PROGRAM Motor_Control
VAR
	Start_Stop_0: Start_Stop;
	Trapizoidal_0: Trapizoidal;
	Trapizoidal_1: Trapizoidal;
	BLINK_0: BLINK;
	R_TRIG_0: R_TRIG;
	
	Timer : BOOL;
END_VAR

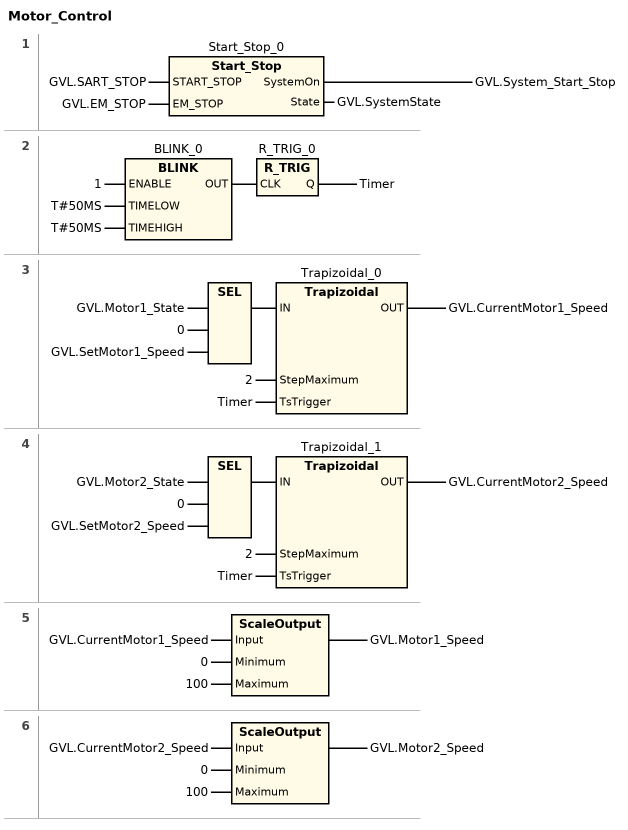
// NETWORK 1
Start_Stop_0(START_STOP := GVL.SART_STOP, EM_STOP := GVL.EM_STOP, State => GVL.SystemState); // Start_Stop
GVL.System_Start_Stop := Start_Stop_0.SystemOn;

// NETWORK 2
BLINK_0(ENABLE := 1, TIMELOW := T#50MS, TIMEHIGH := T#50MS); // BLINK
R_TRIG_0(CLK := BLINK_0.OUT); // R_TRIG
Timer := R_TRIG_0.Q;

// NETWORK 3
Trapizoidal_0(IN := SEL(GVL.Motor1_State, 0, GVL.SetMotor1_Speed), StepMaximum := 2, TsTrigger := Timer); // Trapizoidal
GVL.CurrentMotor1_Speed := Trapizoidal_0.OUT;

// NETWORK 4
Trapizoidal_1(IN := SEL(GVL.Motor2_State, 0, GVL.SetMotor2_Speed), StepMaximum := 2, TsTrigger := Timer); // Trapizoidal
GVL.CurrentMotor2_Speed := Trapizoidal_1.OUT;

// NETWORK 5
GVL.Motor1_Speed := ScaleOutput(Input := GVL.CurrentMotor1_Speed, Minimum := 0, Maximum := 100);

// NETWORK 6
GVL.Motor2_Speed := ScaleOutput(Input := GVL.CurrentMotor2_Speed, Minimum := 0, Maximum := 100);

END_PROGRAM

(* stored: Version 1.1.0.1, ProductVersion 3.1.4024.12
   POU Motor_Control: Id {8528f7c6-565c-49a0-bd8a-e255f0723f91}, SpecialFunc None *)
